// TwinCAT 3 PLC project Tests
// libraries:
//   TcUnit, * (www.tcunit.org)
// project tree:
//   / FB_FilterTests.TcPOU, E_State.TcDUT

// ---- E_State.TcDUT

// :Description: Test-harness state (intentionally collides with Library.E_State to exercise ADR-0005's ambiguous-symbol error path).
TYPE E_State :
(
    Pending := 0,
    Pass := 1,
    Fail := 2
);
END_TYPE

// ---- FB_FilterTests.TcPOU

// :Description: TcUnit suite for FB_Filter.
FUNCTION_BLOCK FB_FilterTests EXTENDS TcUnit.FB_TestSuite
VAR
    filter : FB_Filter;
    state  : E_State;
END_VAR


RollingAverage_passes_known_vector();


METHOD PRIVATE RollingAverage_passes_known_vector

TEST('RollingAverage_passes_known_vector');
AssertEquals_LREAL(Expected := 1.0, Actual := filter.Step(1.0), Delta := 0.001, Message := 'first sample');
TEST_FINISHED();
END_METHOD

END_FUNCTION_BLOCK
